// TIA Portal V17 export
// export: Created 2024-09-27T18:48:47.3413247Z, ExportSetting WithDefaults, DisplayName Totally Integrated Automation Portal, DisplayVersion V17, DisplayName TIA Portal Openness, DisplayVersion V17, DisplayName TIA Portal Version Control Interface, DisplayVersion V17, DisplayName STEP 7 Professional, DisplayVersion V17, DisplayName STEP 7 Safety, DisplayVersion V17, DisplayName WinCC Professional, DisplayVersion V17
DATA_BLOCK "MC_Reset_DB"   // DB10
// stored: AutoNumber true, DBAccessibleFromOPCUA true, InstanceOfName MC_Reset, OfSystemLibElement MC_Reset, OfSystemLibVersion 8.0
"MC_Reset"
   // VAR_INPUT
   //    Axis : TO_Axis;
   //    Execute : Bool;
   //    Restart : Bool;
   // END_VAR
   // VAR_OUTPUT
   //    Done : Bool;
   //    Busy : Bool;
   //    Error : Bool;
   //    ErrorID : Word;
   //    ErrorInfo : Word;
   // END_VAR
   // VAR
   //    FB_ID : DInt;
   // END_VAR
BEGIN
END_DATA_BLOCK
